PROGRAM P_BACnet_Manual
VAR
	dwManual		: DWORD;
	
	rtSet			: R_TRIG;
	rtReset			: R_TRIG;
	
	iSelSet			: INT := 0;
	iSelReset		: INT := 0;
	
	ton_DelayForBACnet		: TON;
	ton_DelayForBACnet_Set	: TON;
END_VAR

//keep BACnet object instance alive
fbBACnet_AV_SL_Manual(Device := Device, bEnablePV := TRUE, bNullPV := FALSE);

//init rising edge detection
rtSet(CLK := bBACnet_SetManual);
rtReset(CLK := bBACnet_ResetManual);


//if rising edge occures
IF rtSet.Q AND NOT bBACnet_ResetManual AND iSelSet = 0 THEN
	//set selector to 10
	iSelSet := 10;
END_IF
IF rtReset.Q AND NOT bBACnet_SetManual AND iSelReset = 0 THEN 
	//set selector to 10
	iSelReset := 10;	
END_IF

CASE iSelSet OF
	0:	//idle
		;	//do nothing
	10:
		fbBACnet_AV_SL_Manual.fPV := DWORD_TO_REAL(2#0001111111111111);
		iSelSet := 20;
	20:
		//dalay for BACnet to catch up PLC
		ton_DelayForBACnet_Set(IN := NOT ton_DelayForBACnet_Set.Q, PT := T#100MS);
		IF ton_DelayForBACnet_Set.Q THEN
			//if fPresentValue and fPV are different
			IF fbBACnet_AV_SL_Manual.fPresentValue <> fbBACnet_AV_SL_Manual.fPV THEN
				//increment fPV by 2#0001000000000000 to force the change of fPresentValue
				fbBACnet_AV_SL_Manual.fPV := fbBACnet_AV_SL_Manual.fPV + DWORD_TO_REAL(2#0001000000000000);
			ELSE
				iSelSet := 30;
			END_IF
		END_IF
	30:
		ton_DelayForBACnet_Set(IN := NOT ton_DelayForBACnet_Set.Q, PT := T#100MS);
		IF ton_DelayForBACnet_Set.Q THEN
			bBACnet_SetManual := FALSE;
			iSelSet := 0;
		END_IF
END_CASE

CASE iSelReset OF
	0:	//idle
		;	//do nothing
	10:
		fbBACnet_AV_SL_Manual.fPV := DWORD_TO_REAL(2#0001000000000000);
		iSelReset := 20;
	20:
		//dalay for BACnet to catch up PLC
		ton_DelayForBACnet(IN := NOT ton_DelayForBACnet.Q, PT := T#100MS);
		IF ton_DelayForBACnet.Q THEN
			//if fPresentValue and fPV are different
			IF fbBACnet_AV_SL_Manual.fPresentValue <> fbBACnet_AV_SL_Manual.fPV THEN
				//increment fPV by 2#0001000000000000 to force the change of fPresentValue
				fbBACnet_AV_SL_Manual.fPV := fbBACnet_AV_SL_Manual.fPV + DWORD_TO_REAL(2#0001000000000000);
			ELSE
				iSelReset := 30;
			END_IF
		END_IF
	30:
		ton_DelayForBACnet(IN := NOT ton_DelayForBACnet.Q, PT := T#100MS);
		IF ton_DelayForBACnet.Q THEN
			bBACnet_ResetManual := FALSE;
			iSelReset := 0;
		END_IF
END_CASE


//read REAL data from BACnet object
//and convert them to DWORD
dwManual := REAL_TO_DWORD(fbBACnet_AV_SL_Manual.fPresentValue);

//assign manual control flags
GVL_IO.arrStreetLamps[1].bManualCtrl := dwManual.0;
GVL_IO.arrStreetLamps[2].bManualCtrl := dwManual.1;
GVL_IO.arrStreetLamps[3].bManualCtrl := dwManual.2;
GVL_IO.arrStreetLamps[4].bManualCtrl := dwManual.3;
GVL_IO.arrStreetLamps[5].bManualCtrl := dwManual.4;
GVL_IO.arrStreetLamps[6].bManualCtrl := dwManual.5;
GVL_IO.arrStreetLamps[7].bManualCtrl := dwManual.6;
GVL_IO.arrStreetLamps[8].bManualCtrl := dwManual.7;
GVL_IO.arrStreetLamps[9].bManualCtrl := dwManual.8;
GVL_IO.arrStreetLamps[10].bManualCtrl := dwManual.9;

END_PROGRAM

(* stored: Version 1.1.0.1, ProductVersion 3.1.4024.5
   POU P_BACnet_Manual: Id {17a4fc6b-b4bf-46ca-a744-d8b1a41d2cba}, SpecialFunc None *)
